// TIA Portal V19 export
// export: Created 2026-08-08T14:07:58.2802551Z, ExportSetting WithDefaults, DisplayName Totally Integrated Automation Portal, DisplayVersion V19, DisplayName TIA Portal Openness, DisplayVersion V19, DisplayName TIA Portal Version Control Interface, DisplayVersion V19, DisplayName STEP 7 Professional, DisplayVersion V19, DisplayName STEP 7 Safety, DisplayVersion V19, DisplayName WinCC Basic/Comfort/Advanced, DisplayVersion V19, DisplayName WinCC Unified, DisplayVersion V19
FUNCTION "ce" : Void   // FC1, LAD
{ S7_Optimized_Access := 'TRUE' }
VERSION : 0.1
// stored: AutoNumber true, IsIECCheckEnabled false, SetENOAutomatically false, UDAEnableTagReadback false
   VAR_INPUT
      in1 : Bool;
      in2 : Int;
      in3 : Int;
      in4 : Int;
      in5 : Bool;
   END_VAR
   VAR_OUTPUT
      out1 : Bool;
      out2 : Int;
      out3 : Int;
   END_VAR
BEGIN

REGION Network 1
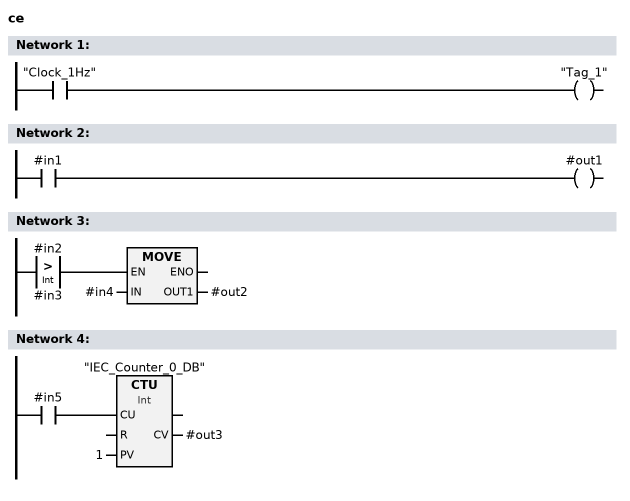
   RUNG wire#powerrail
      Contact( "Clock_1Hz" )
      Coil( "Tag_1" )
   END_RUNG
   // the same network as SCL:
   "Tag_1" := "Clock_1Hz";
END_REGION

REGION Network 2
   RUNG wire#powerrail
      Contact( #in1 )
      Coil( #out1 )
   END_RUNG
   // the same network as SCL:
   #out1 := #in1;
END_REGION

REGION Network 3
   RUNG wire#powerrail
      { S7_Templates := "SrcType := Int" } GT_Contact(in1 := #in2, in2 := #in3)
      Move(in := #in4, out1 => #out2)
   END_RUNG
   // the same network as SCL:
   IF #in2 > #in3 THEN #out2 := #in4; END_IF;
END_REGION

REGION Network 4
   RUNG wire#powerrail
      Contact( #in5 )
      { S7_Templates := "value_type := Int" } "IEC_Counter_0_DB".CTU(r :=, pv := 1, cv => #out3)
   END_RUNG
   // the same network as SCL:
   "IEC_Counter_0_DB".CTU(CU := #in5, PV := 1, CV => #out3);
END_REGION
END_FUNCTION
